// TwinCAT 3 PLC project OOB
// ProgramVersion: 3.1.4026.20
// libraries:
//   Tc2_ControllerToolbox, * (Beckhoff Automation GmbH)
//   Tc2_Standard, * (Beckhoff Automation GmbH)
//   Tc2_System, * (Beckhoff Automation GmbH)
// project tree:
//   FBs/ FB_Lampe.TcPOU, FB_Manager.TcPOU, FB_Valve.TcPOU
//   GVLs/ Process.TcGVL
//   / PlcTask.TcTTO
//   POUs/ MAIN.TcPOU, PRG_System.TcPOU

CONFIGURATION OOB
    RESOURCE PLC ON TwinCAT3
        TASK PlcTask(INTERVAL := T#10ms, PRIORITY := 20);
        PROGRAM MAIN WITH PlcTask : MAIN;
    END_RESOURCE
END_CONFIGURATION

// ---- GVLs/Process.TcGVL
{attribute 'qualified_only'}
VAR_GLOBAL
	// Defaulting auto mode.
	eCtrlMode:				E_CTRL_MODE:=E_CTRL_MODE.eCTRL_MODE_ACTIVE;
END_VAR

// ---- POUs/MAIN.TcPOU
PROGRAM MAIN
VAR
	fbValveHotWater:	FB_Valve;
	fbValveColdWater:	FB_Valve;
	fbValveBypass:		FB_Valve;
	bValve:		BOOL;
END_VAR

fbValveHotWater(bIn:=TRUE, bOut=>bValve);

END_PROGRAM

// ---- FBs/FB_Valve.TcPOU
FUNCTION_BLOCK FB_Valve
VAR_INPUT
	bIn:				BOOL;
END_VAR
VAR_OUTPUT
	bOut AT %Q*:		BOOL;
END_VAR
VAR
	tOn:				TON;
	tOff:				TOF;
	tOnTime:			TIME;
	tOffTime:			TIME;
	bReqState:			BOOL;
END_VAR

CASE Process.eCtrlMode OF
	
	(*
	 *	Idle mode: This mode offers no control.
	 *)
	E_CTRL_MODE.eCTRL_MODE_IDLE:
		tOn(IN:=FALSE);
		tOff(IN:=FALSE);
		bOut:=FALSE;
		
	(*
	 *	Manual mode: This mode offers direct control from the admin
	 *	this has no delay.
	 *)
	E_CTRL_MODE.eCTRL_MODE_MANUAL:
		tOn(IN:=FALSE);
		tOff(IN:=FALSE);
		bOut:=bIn;
		
	(*
	 *	Auto mode: This mode allows for the FB to be set up with
	 *	ON-delay and OFF-delay
	 *)
	E_CTRL_MODE.eCTRL_MODE_ACTIVE:
		tOn (IN:=bIn, PT:=tOnTime);
		tOff (IN:=bIn, PT:=tOffTime);
		CASE TO_INT(bOut) OF
			0:
				IF tOn.Q THEN
					bOut:=TRUE;
				END_IF
			1:
				IF NOT tOff.Q THEN
					bOut:=FALSE;
				END_IF
		END_CASE
ELSE
	(*
	 *	Fail-state or invalid mode: Valve-default is off
	 *)
	tOn(IN:=FALSE);
	tOff(IN:=FALSE);
	bOut:=FALSE;
END_CASE

METHOD Init : BOOL
VAR_INPUT
	tOnTimeInit:	TIME:=T#10S;
	tOffTimeInit:	TIME:=T#10s;
END_VAR
tOnTime:=tOnTimeInit;
tOffTime:=tOffTimeInit;
Init:=TRUE;
END_METHOD

END_FUNCTION_BLOCK

// ---- FBs/FB_Lampe.TcPOU
FUNCTION_BLOCK FB_Lampe
VAR
    bOn : BOOL;
    bInit : BOOL := FALSE;
END_VAR

METHOD Init
VAR_INPUT
    fbManager : REFERENCE TO FB_Manager;
END_VAR
IF NOT bInit THEN
    fbManager.Register(THIS);
    bInit := TRUE;
END_IF
END_METHOD

END_FUNCTION_BLOCK

// ---- FBs/FB_Manager.TcPOU
FUNCTION_BLOCK FB_Manager
VAR
    arrLamper : ARRAY[1..10] OF POINTER TO FB_Lampe;
    iCount    : INT := 0;
END_VAR

METHOD Register
VAR_INPUT
    pLampe : POINTER TO FB_Lampe;
END_VAR
IF iCount < 10 THEN
    iCount := iCount + 1;
    arrLamper[iCount] := pLampe;
END_IF
END_METHOD

METHOD SlukAlle
VAR
    i : INT;
END_VAR
FOR i := 1 TO iCount DO
    arrLamper[i]^.bOn := FALSE;
END_FOR
END_METHOD

END_FUNCTION_BLOCK

// ---- POUs/PRG_System.TcPOU
PROGRAM PRG_System
VAR
    fbManager : FB_Manager;

    lampe1 : FB_Lampe;
    lampe2 : FB_Lampe;
END_VAR

lampe1.Init(fbManager);
lampe2.Init(fbManager);

END_PROGRAM
